(* CODESYS project Lift Uitgewerkt - Ladder SFC V02.project

Project tree, tasks and I/O mapping:
  Device : CODESYS Control Win V3, 3S - Smart Software Solutions GmbH, version 3.5.16.70
    application Application
      libraries: Standard, * (System)
      task MainTask (cyclic, interval t#20ms, priority 1) calls Aandrijving, BenedenDeur, BovenDeur, Controller, Hoofdprogramma, Simulatie
      visualisation Visualization
  Lift Besturing/
    program Hoofdprogramma [SFC]
    program Aandrijving [SFC]
    program Controller [LD]
    program BovenDeur [SFC]
    program BenedenDeur [SFC]
  global variables GVL
  image pool ImagePool
  5ce3da45-db07-42e7-a21c-a00fff4ed8f6|C:\Users\Gerard\Desktop\MensenInLift.PNG
  5ce3da45-db07-42e7-a21c-a00fff4ed8f6|C:\Users\Gerard\Desktop\LiftDeur.PNG
  5ce3da45-db07-42e7-a21c-a00fff4ed8f6|C:\Users\Gerard\Desktop\Liftaandrijving.PNG
  5ce3da45-db07-42e7-a21c-a00fff4ed8f6|C:\Users\Gerard\Desktop\LiftDeurAandrijving.PNG
  Lift Simualtie/
    program Simulatie [ST]
  text list GlobalTextList
*)

// GVL
VAR_GLOBAL
	Ix_BovenOproepKooi					: BOOL;
	Ix_BenedenOproepKooi				: BOOL;
	Ix_KooiGaNaarBoven					: BOOL;
	Ix_KooiGaNaarBeneden				: BOOL;
	Ix_KooiBoven						: BOOL;
	Ix_KooiBeneden						: BOOL;
	Qx_AandrijvingOmhoog				: BOOL;
	Qx_AandrijvingOmlaag				: BOOL;
	
	
	Ix_BenedenDeurOpen					: BOOL;
	Ix_BenedenDeurGesloten				: BOOL;
	Qx_BenedenDeurAandrijvingOpen		: BOOL;
	Qx_BenedenDeurAandrijvingSluiten	: BOOL;
	
	Ix_BovenDeurOpen					: BOOL;
	Ix_BovenDeurGesloten				: BOOL;
	Qx_BovenDeurAandrijvingOpen			: BOOL;
	Qx_BovenDeurAandrijvingSluiten		: BOOL;
	
	
END_VAR

// Lift Besturing/Aandrijving
// Programma		: Aandrijving
// Project			: Lift
// Doel				: Aandrijven van de lift kooi
// Auteur			: Gerard Harkema
// Versie			: 1.0
// Datum			: 15 oktober 2015

PROGRAM Aandrijving
VAR_INPUT
	Mx_StartAandrijvingOmhoog: BOOL;
	Mx_StartAandrijvingOmlaag: BOOL;
END_VAR

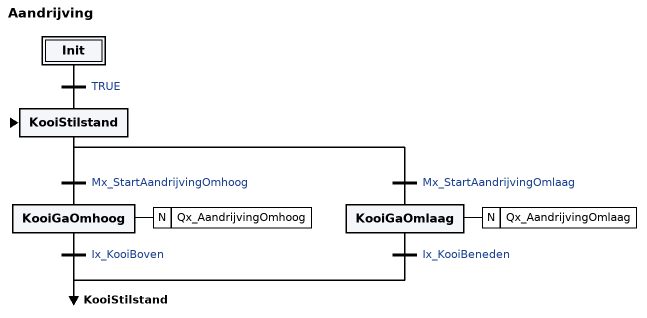
INITIAL_STEP Init:
END_STEP
TRANSITION FROM Init TO KooiStilstand
    := TRUE;
END_TRANSITION
STEP KooiStilstand:
END_STEP
TRANSITION FROM KooiStilstand TO KooiGaOmhoog
    := Mx_StartAandrijvingOmhoog;
END_TRANSITION
STEP KooiGaOmhoog:
    Qx_AandrijvingOmhoog(N);
END_STEP
TRANSITION FROM KooiGaOmhoog TO KooiStilstand
    := Ix_KooiBoven;
END_TRANSITION
TRANSITION FROM KooiStilstand TO KooiGaOmlaag
    := Mx_StartAandrijvingOmlaag;
END_TRANSITION
STEP KooiGaOmlaag:
    Qx_AandrijvingOmlaag(N);
END_STEP
TRANSITION FROM KooiGaOmlaag TO KooiStilstand
    := Ix_KooiBeneden;
END_TRANSITION

END_PROGRAM

// Lift Besturing/BenedenDeur
// Programma		: BenedenDeur
// Project			: Lift
// Doel				: Aandrijving van de benedendeur
// Auteur			: Gerard Harkema
// Versie			: 1.0
// Datum			: 15 oktober 2015


PROGRAM BenedenDeur
VAR_INPUT
	Mx_BenedenDeurSluiten: BOOL;
	Mx_BenedenDeurOpenen: BOOL;
END_VAR

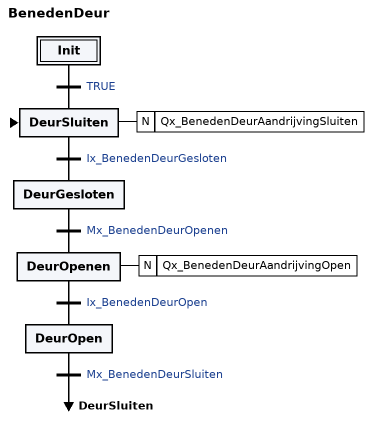
INITIAL_STEP Init:
END_STEP
TRANSITION FROM Init TO DeurSluiten
    := TRUE;
END_TRANSITION
STEP DeurSluiten:
    Qx_BenedenDeurAandrijvingSluiten(N);
END_STEP
TRANSITION FROM DeurSluiten TO DeurGesloten
    := Ix_BenedenDeurGesloten;
END_TRANSITION
STEP DeurGesloten:
END_STEP
TRANSITION FROM DeurGesloten TO DeurOpenen
    := Mx_BenedenDeurOpenen;
END_TRANSITION
STEP DeurOpenen:
    Qx_BenedenDeurAandrijvingOpen(N);
END_STEP
TRANSITION FROM DeurOpenen TO DeurOpen
    := Ix_BenedenDeurOpen;
END_TRANSITION
STEP DeurOpen:
END_STEP
TRANSITION FROM DeurOpen TO DeurSluiten
    := Mx_BenedenDeurSluiten;
END_TRANSITION

END_PROGRAM

// Lift Besturing/BovenDeur
// Programma		: BovenDeur
// Project			: Lift
// Doel				: Aandrijving van de bovendeur
// Auteur			: Gerard Harkema
// Versie			: 1.0
// Datum			: 15 oktober 2015

PROGRAM BovenDeur
VAR_INPUT
	Mx_BovenDeurSluiten: BOOL;
	Mx_BovenDeurOpenen: BOOL;
END_VAR

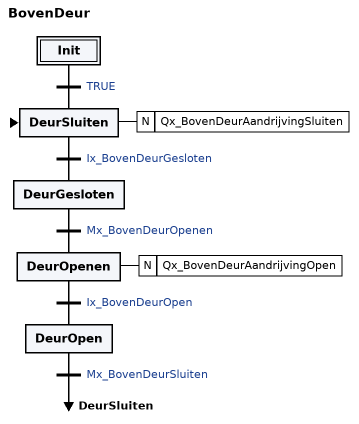
INITIAL_STEP Init:
END_STEP
TRANSITION FROM Init TO DeurSluiten
    := TRUE;
END_TRANSITION
STEP DeurSluiten:
    Qx_BovenDeurAandrijvingSluiten(N);
END_STEP
TRANSITION FROM DeurSluiten TO DeurGesloten
    := Ix_BovenDeurGesloten;
END_TRANSITION
STEP DeurGesloten:
END_STEP
TRANSITION FROM DeurGesloten TO DeurOpenen
    := Mx_BovenDeurOpenen;
END_TRANSITION
STEP DeurOpenen:
    Qx_BovenDeurAandrijvingOpen(N);
END_STEP
TRANSITION FROM DeurOpenen TO DeurOpen
    := Ix_BovenDeurOpen;
END_TRANSITION
STEP DeurOpen:
END_STEP
TRANSITION FROM DeurOpen TO DeurSluiten
    := Mx_BovenDeurSluiten;
END_TRANSITION

END_PROGRAM

// Lift Besturing/Controller
// Programma		: Controller
// Project			: Lift
// Doel				: Afhandeling signalen voor de liftbesturing
// Auteur			: Gerard Harkema
// Versie			: 1.0
// Datum			: 15 oktober 2015
PROGRAM Controller
VAR
	Mx_GaOmhoog: BOOL;
	Mx_GaOmlaag: BOOL;

END_VAR

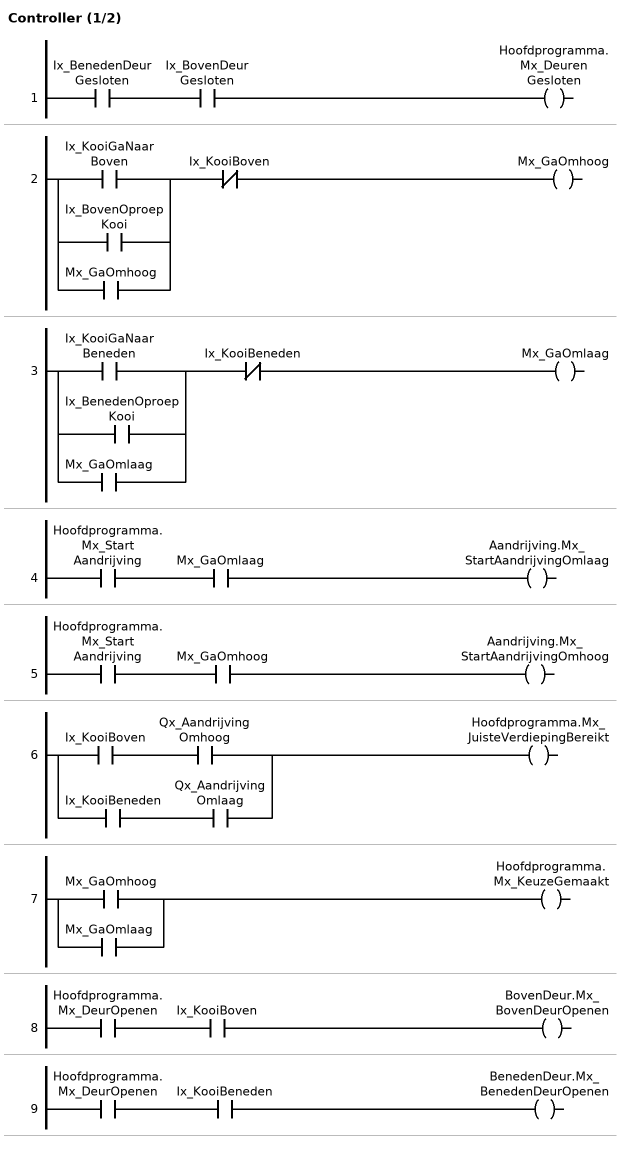
// NETWORK 1
Hoofdprogramma.Mx_DeurenGesloten := Ix_BenedenDeurGesloten AND Ix_BovenDeurGesloten;

// NETWORK 2
Mx_GaOmhoog := (Ix_KooiGaNaarBoven OR Ix_BovenOproepKooi OR Mx_GaOmhoog) AND NOT Ix_KooiBoven;

// NETWORK 3
Mx_GaOmlaag := (Ix_KooiGaNaarBeneden OR Ix_BenedenOproepKooi OR Mx_GaOmlaag) AND NOT Ix_KooiBeneden;

// NETWORK 4
Aandrijving.Mx_StartAandrijvingOmlaag := Hoofdprogramma.Mx_StartAandrijving AND Mx_GaOmlaag;

// NETWORK 5
Aandrijving.Mx_StartAandrijvingOmhoog := Hoofdprogramma.Mx_StartAandrijving AND Mx_GaOmhoog;

// NETWORK 6
Hoofdprogramma.Mx_JuisteVerdiepingBereikt := Ix_KooiBoven AND Qx_AandrijvingOmhoog OR Ix_KooiBeneden AND Qx_AandrijvingOmlaag;

// NETWORK 7
Hoofdprogramma.Mx_KeuzeGemaakt := Mx_GaOmhoog OR Mx_GaOmlaag;

// NETWORK 8
BovenDeur.Mx_BovenDeurOpenen := Hoofdprogramma.Mx_DeurOpenen AND Ix_KooiBoven;

// NETWORK 9
BenedenDeur.Mx_BenedenDeurOpenen := Hoofdprogramma.Mx_DeurOpenen AND Ix_KooiBeneden;

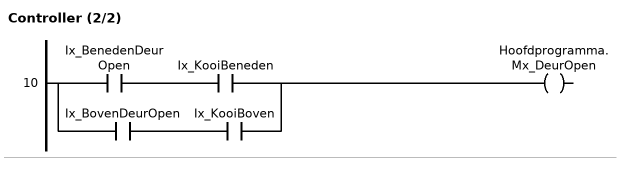
// NETWORK 10
Hoofdprogramma.Mx_DeurOpen := Ix_BenedenDeurOpen AND Ix_KooiBeneden OR Ix_BovenDeurOpen AND Ix_KooiBoven;

END_PROGRAM

// Lift Besturing/Hoofdprogramma
// Programma		: Hoofdprograamma
// Project			: Lift
// Doel				: Centrale besturing van de liftinstallatie
// Auteur			: Gerard Harkema
// Versie			: 1.0
// Datum			: 15 oktober 2015

PROGRAM Hoofdprogramma
VAR_INPUT
	Mx_JuisteVerdiepingBereikt: BOOL;
	Mx_KeuzeGemaakt: BOOL;
	Mx_DeurOpen: BOOL;
	Mx_DeurenGesloten: BOOL;
	Mx_StartAandrijving: BOOL;
	Mx_DeurOpenen: BOOL;
END_VAR

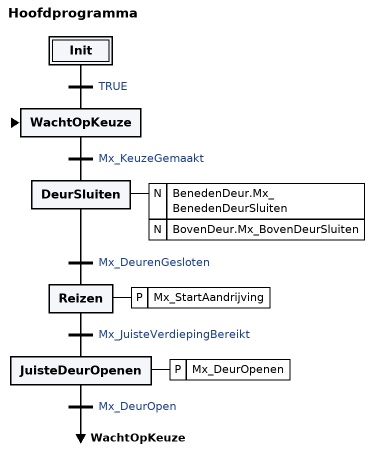
INITIAL_STEP Init:
END_STEP
TRANSITION FROM Init TO WachtOpKeuze
    := TRUE;
END_TRANSITION
STEP WachtOpKeuze:
END_STEP
TRANSITION FROM WachtOpKeuze TO DeurSluiten
    := Mx_KeuzeGemaakt;
END_TRANSITION
STEP DeurSluiten:
    BenedenDeur.Mx_BenedenDeurSluiten(N);
    BovenDeur.Mx_BovenDeurSluiten(N);
END_STEP
TRANSITION FROM DeurSluiten TO Reizen
    := Mx_DeurenGesloten;
END_TRANSITION
STEP Reizen:
    Mx_StartAandrijving(P);
END_STEP
TRANSITION FROM Reizen TO JuisteDeurOpenen
    := Mx_JuisteVerdiepingBereikt;
END_TRANSITION
STEP JuisteDeurOpenen:
    Mx_DeurOpenen(P);
END_STEP
TRANSITION FROM JuisteDeurOpenen TO WachtOpKeuze
    := Mx_DeurOpen;
END_TRANSITION

END_PROGRAM

// Lift Simualtie/Simulatie
// Programma		: Simulatie
// Project			: Lift
// Doel				: Simulatie functies voor de lift
// Auteur			: Gerard Harkema
// Versie			: 1.0
// Datum			: 15 oktober 2015

PROGRAM Simulatie
VAR
	FB_PulsgeverTimer					: TON;
	Mw_PulsgeverTimerPT					: TIME := T#10MS;
	Mx_PulsLiftAandrijving				: BOOL;
	Mx_Pulsgever						: BOOL;
	Mw_PelsgeverTimerET					: TIME;
	FB_SnelheidLift						: CTU;
	Mw_SnelheidLiftPV					: WORD := 4;
	Mw_SnelheidLiftCV					: WORD;

	Mw_PositieLiftInv					: INT := 0;
	Mw_PositieLift						: INT := 0;
	Mw_LiftBenedenCountValue			: INT := 250;

	Mw_BenedenPositieDeur				: INT := 0;
	Mw_BenedenPositieDeurCountValue		: INT := 100;

	Mw_BovenPositieDeur					: INT := 0;
	Mw_BovenPositieDeurCountValue		: INT := 100;

END_VAR

// Puls gever voor de bewegings simualties

FB_PulsgeverTimer(IN:= (NOT Mx_Pulsgever),PT:= Mw_PulsgeverTimerPT ,Q => Mx_Pulsgever, ET => Mw_PelsgeverTimerET);

//*********************************************
//                 Lift
//*********************************************

// Snelheid lift
FB_SnelheidLift(CU := Mx_Pulsgever, RESET := Mx_PulsLiftAandrijving, PV := Mw_SnelheidLiftPV, Q => Mx_PulsLiftAandrijving, CV => Mw_SnelheidLiftCV);

// Detectie lift is boven
IF (Mw_PositieLiftInv >= Mw_LiftBenedenCountValue) THEN
	GVL.Ix_KooiBoven := TRUE;
ELSE
	GVL.Ix_KooiBoven := FALSE;	
END_IF
  

// Detectie lift is beneden
IF(Mw_PositieLiftInv <= 0) THEN
	GVL.Ix_KooiBeneden := TRUE;
ELSE
	GVL.Ix_KooiBeneden := FALSE;	
END_IF


// Reizen lift omhoog
IF(GVL.Qx_AandrijvingOmhoog AND Mx_PulsLiftAandrijving AND (NOT GVL.Ix_KooiBoven)) THEN
	Mw_PositieLiftInv := Mw_PositieLiftInv + 5;
END_IF

// Reizen lift omlaag
IF(GVL.Qx_AandrijvingOmlaag AND Mx_PulsLiftAandrijving AND (NOT GVL.Ix_KooiBeneden)) THEN
	Mw_PositieLiftInv := Mw_PositieLiftInv - 5;
END_IF

Mw_PositieLift := Mw_LiftBenedenCountValue - Mw_PositieLiftInv;


// Inactief maken oproepknoppen
IF GVL.Ix_KooiBoven THEN
 Ix_BovenOproepKooi := FALSE;
END_IF

IF GVL.Ix_KooiBoven THEN
 Ix_KooiGaNaarBoven := FALSE;
END_IF


IF GVL.Ix_KooiBeneden THEN
 Ix_BenedenOproepKooi := FALSE;
END_IF

IF GVL.Ix_KooiBeneden THEN
 Ix_KooiGaNaarBeneden := FALSE;
END_IF
 

//*********************************************
//                 Benedendeur
//*********************************************

// Detectie Benedendeur is open
IF (Mw_BenedenPositieDeur >= Mw_BenedenPositieDeurCountValue) THEN
	GVL.Ix_BenedenDeurOpen := TRUE;
ELSE
	GVL.Ix_BenedenDeurOpen := FALSE;	
END_IF
  

// Detectie Benedendeur is gesloten
IF(Mw_BenedenPositieDeur <= 0) THEN
	GVL.Ix_BenedenDeurGesloten := TRUE;
ELSE
	GVL.Ix_BenedenDeurGesloten := FALSE;	
END_IF


// Benedendeur openen
IF(GVL.Qx_BenedenDeurAandrijvingOpen AND Mx_PulsLiftAandrijving AND (NOT GVL.Ix_BenedenDeurOpen)) THEN
	Mw_BenedenPositieDeur := Mw_BenedenPositieDeur + 5;
END_IF

// Benedendeur sluiten
IF(GVL.Qx_BenedenDeurAandrijvingSluiten AND Mx_PulsLiftAandrijving AND (NOT GVL.Ix_BenedenDeurGesloten)) THEN
	Mw_BenedenPositieDeur := Mw_BenedenPositieDeur - 5;
END_IF

//*********************************************
//                 Bovendeur
//*********************************************

// Detectie bovendeur is open
IF (Mw_BovenPositieDeur >= Mw_BovenPositieDeurCountValue) THEN
	GVL.Ix_BovenDeurOpen := TRUE;
ELSE
	GVL.Ix_BovenDeurOpen := FALSE;	
END_IF
  

// Detectie bovendeur is gesloten
IF(Mw_BovenPositieDeur <= 0) THEN
	GVL.Ix_BovenDeurGesloten := TRUE;
ELSE
	GVL.Ix_BovenDeurGesloten := FALSE;	
END_IF


// Bovendeur openen
IF(GVL.Qx_BovenDeurAandrijvingOpen AND Mx_PulsLiftAandrijving AND (NOT GVL.Ix_BovenDeurOpen)) THEN
	Mw_BovenPositieDeur := Mw_BovenPositieDeur + 5;
END_IF

// Bovendeur sluiten
IF(GVL.Qx_BovenDeurAandrijvingSluiten AND Mx_PulsLiftAandrijving AND (NOT GVL.Ix_BovenDeurGesloten)) THEN
	Mw_BovenPositieDeur := Mw_BovenPositieDeur - 5;
END_IF

END_PROGRAM

// Device/Application/Visualization
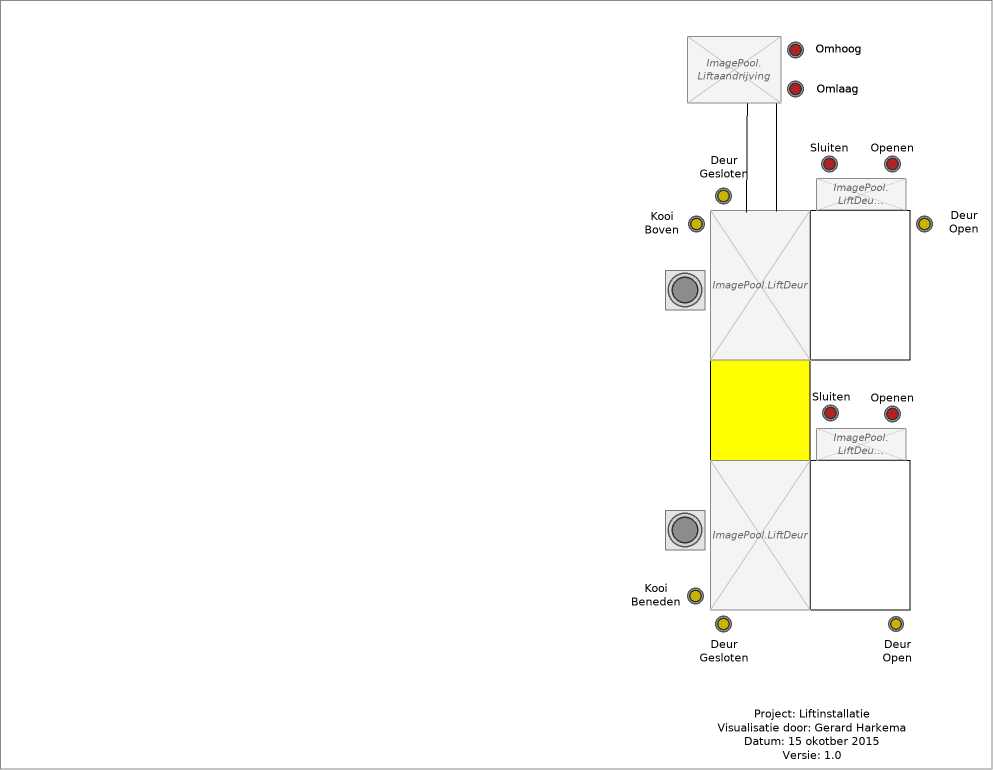
VISUALIZATION Visualization  // 993x770
    Rectangle (810,460 100x150)
    Rectangle (810,210 100x150)
    Rectangle (710,210 100x400)
    PushSwitch (665,270 40x40), tooltip "Oproep Boven", variable: Ix_BovenOproepKooi, behaviour: TOGGLE, style: Switch-PushSwitch-Gray
    PushSwitch (665,510 40x40), tooltip "Oproep Beneden", variable: Ix_BenedenOproepKooi, behaviour: TOGGLE, style: Switch-PushSwitch-Gray
    Group (710,210 100x150)
        p2738717112: Simulatie.Mw_PositieLift
        Rectangle (0,0 100x150)
        Image (6,0 89x150), image: ImagePool.MensenInLift
        PushSwitch (5,100 30x30), tooltip "Ga naar beneden", variable: Ix_KooiGaNaarBeneden, behaviour: TOGGLE, style: Switch-PushSwitch-Gray
        PushSwitch (5,60 30x30), tooltip "Ga naar Boven", variable: Ix_KooiGaNaarBoven, behaviour: TOGGLE, style: Switch-PushSwitch-Gray
    Rectangle (710,210 100x150)
    Image (716,210 89x150), image: ImagePool.MensenInLift
    PushSwitch (715,310 30x30), tooltip "Ga naar beneden", variable: Ix_KooiGaNaarBeneden, behaviour: TOGGLE, style: Switch-PushSwitch-Gray
    PushSwitch (715,270 30x30), tooltip "Ga naar Boven", variable: Ix_KooiGaNaarBoven, behaviour: TOGGLE, style: Switch-PushSwitch-Gray
    Lamp1 (714,186 19x20), variable: Ix_BovenDeurGesloten, style: Lamp-Lamp1-Yellow
    Lamp1 (915,214 19x20), variable: Ix_BovenDeurOpen, style: Lamp-Lamp1-Yellow
    Lamp1 (687,214 19x20), variable: Ix_KooiBoven, style: Lamp-Lamp1-Yellow
    Lamp1 (686,586 19x20), variable: Ix_KooiBeneden, style: Lamp-Lamp1-Yellow
    Lamp1 (714,614 19x20), variable: Ix_BenedenDeurGesloten, style: Lamp-Lamp1-Yellow
    Lamp1 (887,614 18x20), variable: Ix_BenedenDeurOpen, style: Lamp-Lamp1-Yellow
    Label (682,152 84x30), "Deur Gesloten"
    Label (937,207 54x30), "Deur Open"
    Label (640,208 44x30), "Kooi Boven"
    Label (629,580 54x30), "Kooi Beneden"
    Label (693,636 62x30), "Deur Gesloten"
    Label (875,636 45x30), "Deur Open"
    Group (710,210 100x150)
        p3560616238: Simulatie.Mw_BovenPositieDeur
        Rectangle (0,0 100x150)
        Image (0,0 100x150), image: ImagePool.LiftDeur
    Group (710,460 100x150)
        p3560616238: Simulatie.Mw_BenedenPositieDeur
        Rectangle (0,0 100x150)
        Image (0,0 100x150), image: ImagePool.LiftDeur
    Line (747,83) (746,212)
    Line (776,82) (776,211)
    Group (687,34 182x70)
        Image (0,2 94x67), image: ImagePool.Liftaandrijving
        Lamp1 (99,6 19x20), variable: Qx_AandrijvingOmhoog, style: Lamp-Lamp1-Red
        Lamp1 (99,45 19x20), variable: Qx_AandrijvingOmlaag, style: Lamp-Lamp1-Red
        Label (121,0 61x30), "Omhoog"
        Label (123,40 55x30), "Omlaag"
    Image (687,36 94x67), image: ImagePool.Liftaandrijving
    Lamp1 (786,40 19x20), variable: Qx_AandrijvingOmhoog, style: Lamp-Lamp1-Red
    Lamp1 (786,79 19x20), variable: Qx_AandrijvingOmlaag, style: Lamp-Lamp1-Red
    Label (808,34 61x30), "Omhoog"
    Label (810,74 55x30), "Omlaag"
    Group (816,154 90x56)
        Image (0,24 90x32), image: ImagePool.LiftDeurAandrijving
        Lamp1 (4,0 19x20), variable: Qx_BovenDeurAandrijvingSluiten, style: Lamp-Lamp1-Red
        Lamp1 (67,0 19x20), variable: Qx_BovenDeurAandrijvingOpen, style: Lamp-Lamp1-Red
    Image (816,178 90x32), image: ImagePool.LiftDeurAandrijving
    Lamp1 (820,154 19x20), variable: Qx_BovenDeurAandrijvingSluiten, style: Lamp-Lamp1-Red
    Lamp1 (883,154 19x20), variable: Qx_BovenDeurAandrijvingOpen, style: Lamp-Lamp1-Red
    Group (816,403 90x57)
        Image (0,25 90x32), image: ImagePool.LiftDeurAandrijving
        Lamp1 (5,0 19x20), variable: Qx_BenedenDeurAandrijvingSluiten, style: Lamp-Lamp1-Red
        Lamp1 (67,1 19x20), variable: Qx_BenedenDeurAandrijvingOpen, style: Lamp-Lamp1-Red
    Image (816,428 90x32), image: ImagePool.LiftDeurAandrijving
    Lamp1 (821,403 19x20), variable: Qx_BenedenDeurAandrijvingSluiten, style: Lamp-Lamp1-Red
    Lamp1 (883,404 19x20), variable: Qx_BenedenDeurAandrijvingOpen, style: Lamp-Lamp1-Red
    Label (812,382 39x30), "Sluiten"
    Label (810,133 39x30), "Sluiten"
    Label (867,383 51x30), "Openen"
    Label (867,133 51x30), "Openen"
    Label (712,701 200x67), "Project: Liftinstallatie Visualisatie door: Gerard Harkema Datum: 15 okotber 2015 Versie: 1.0"
END_VISUALIZATION
